// TIA Portal V20 export
FUNCTION_BLOCK "EventsPFE_Recipe"   // FB125, LAD
// stored: MemoryReserve 100, Namespace Unit1.Em7, SetENOAutomatically false
   VAR
      data : Array[1..100] of LReal;
   END_VAR
BEGIN

REGION Network 1: PDR Data21 Recipe - Hot Press Right Press Pressure
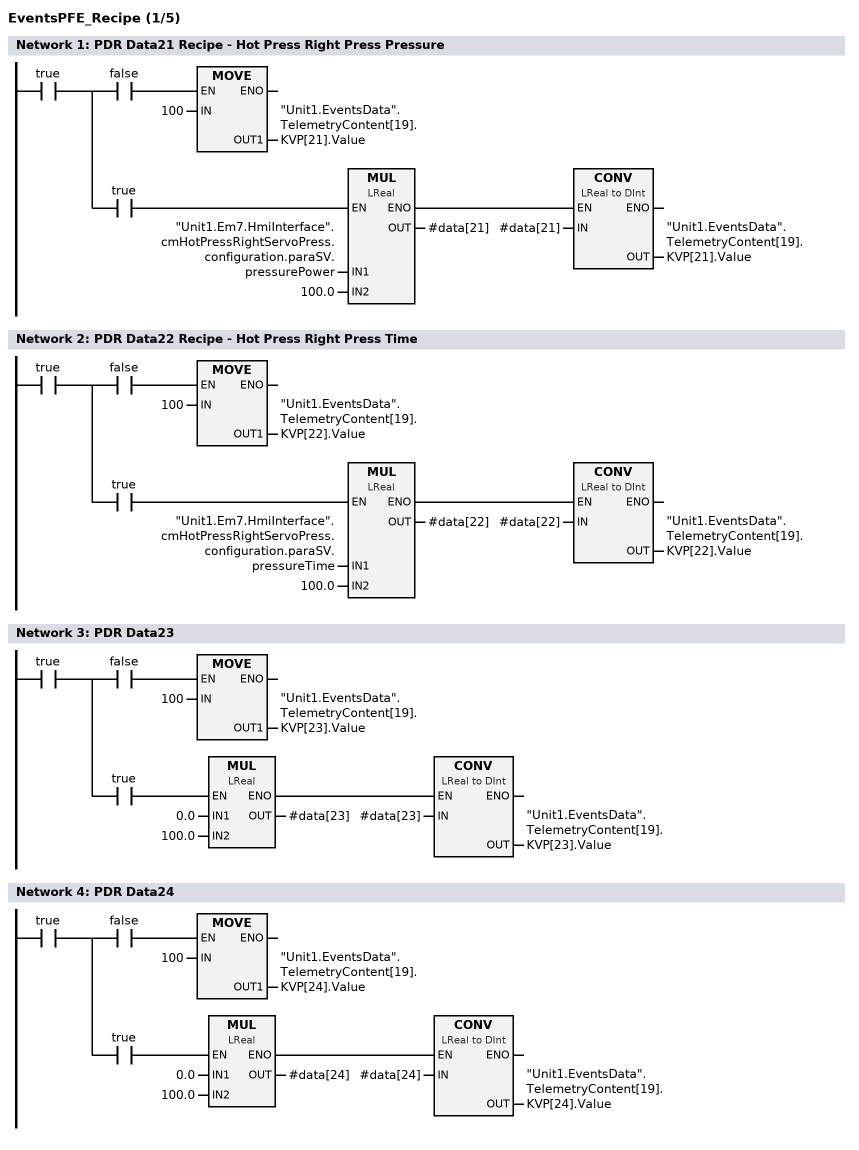
   RUNG wire#powerrail
      Contact( true )
      wire#w1
      Contact( false )
      Move(in := 100, out1 => "Unit1.EventsData".TelemetryContent[19].KVP[21].Value)
   END_RUNG
   RUNG wire#w1
      Contact( true )
      { S7_Templates := "SrcType := LReal" } Mul(in1 := "Unit1.Em7.HmiInterface".cmHotPressRightServoPress.configuration.paraSV.pressurePower, in2 := 100.0, out => #data[21])
      { S7_Templates := "[SrcType := LReal, DestType := DInt]" } Convert(in := #data[21], out => "Unit1.EventsData".TelemetryContent[19].KVP[21].Value)
   END_RUNG
   // the same network as SCL:
   IF true AND false THEN "Unit1.EventsData".TelemetryContent[19].KVP[21].Value := 100; END_IF;
   IF true AND true THEN
       #data[21] := "Unit1.Em7.HmiInterface".cmHotPressRightServoPress.configuration.paraSV.pressurePower * 100.0;
       "Unit1.EventsData".TelemetryContent[19].KVP[21].Value := LREAL_TO_DINT(#data[21]);
   END_IF;
END_REGION

REGION Network 2: PDR Data22 Recipe - Hot Press Right Press Time
   RUNG wire#powerrail
      Contact( true )
      wire#w1
      Contact( false )
      Move(in := 100, out1 => "Unit1.EventsData".TelemetryContent[19].KVP[22].Value)
   END_RUNG
   RUNG wire#w1
      Contact( true )
      { S7_Templates := "SrcType := LReal" } Mul(in1 := "Unit1.Em7.HmiInterface".cmHotPressRightServoPress.configuration.paraSV.pressureTime, in2 := 100.0, out => #data[22])
      { S7_Templates := "[SrcType := LReal, DestType := DInt]" } Convert(in := #data[22], out => "Unit1.EventsData".TelemetryContent[19].KVP[22].Value)
   END_RUNG
   // the same network as SCL:
   IF true AND false THEN "Unit1.EventsData".TelemetryContent[19].KVP[22].Value := 100; END_IF;
   IF true AND true THEN
       #data[22] := "Unit1.Em7.HmiInterface".cmHotPressRightServoPress.configuration.paraSV.pressureTime * 100.0;
       "Unit1.EventsData".TelemetryContent[19].KVP[22].Value := LREAL_TO_DINT(#data[22]);
   END_IF;
END_REGION

REGION Network 3: PDR Data23
   RUNG wire#powerrail
      Contact( true )
      wire#w1
      Contact( false )
      Move(in := 100, out1 => "Unit1.EventsData".TelemetryContent[19].KVP[23].Value)
   END_RUNG
   RUNG wire#w1
      Contact( true )
      { S7_Templates := "SrcType := LReal" } Mul(in1 := 0.0, in2 := 100.0, out => #data[23])
      { S7_Templates := "[SrcType := LReal, DestType := DInt]" } Convert(in := #data[23], out => "Unit1.EventsData".TelemetryContent[19].KVP[23].Value)
   END_RUNG
   // the same network as SCL:
   IF true AND false THEN "Unit1.EventsData".TelemetryContent[19].KVP[23].Value := 100; END_IF;
   IF true AND true THEN
       #data[23] := 0.0 * 100.0;
       "Unit1.EventsData".TelemetryContent[19].KVP[23].Value := LREAL_TO_DINT(#data[23]);
   END_IF;
END_REGION

REGION Network 4: PDR Data24
   RUNG wire#powerrail
      Contact( true )
      wire#w1
      Contact( false )
      Move(in := 100, out1 => "Unit1.EventsData".TelemetryContent[19].KVP[24].Value)
   END_RUNG
   RUNG wire#w1
      Contact( true )
      { S7_Templates := "SrcType := LReal" } Mul(in1 := 0.0, in2 := 100.0, out => #data[24])
      { S7_Templates := "[SrcType := LReal, DestType := DInt]" } Convert(in := #data[24], out => "Unit1.EventsData".TelemetryContent[19].KVP[24].Value)
   END_RUNG
   // the same network as SCL:
   IF true AND false THEN "Unit1.EventsData".TelemetryContent[19].KVP[24].Value := 100; END_IF;
   IF true AND true THEN
       #data[24] := 0.0 * 100.0;
       "Unit1.EventsData".TelemetryContent[19].KVP[24].Value := LREAL_TO_DINT(#data[24]);
   END_IF;
END_REGION

REGION Network 5: PDR Data25 Recipe - Hot Press Right Upper1 Temperature
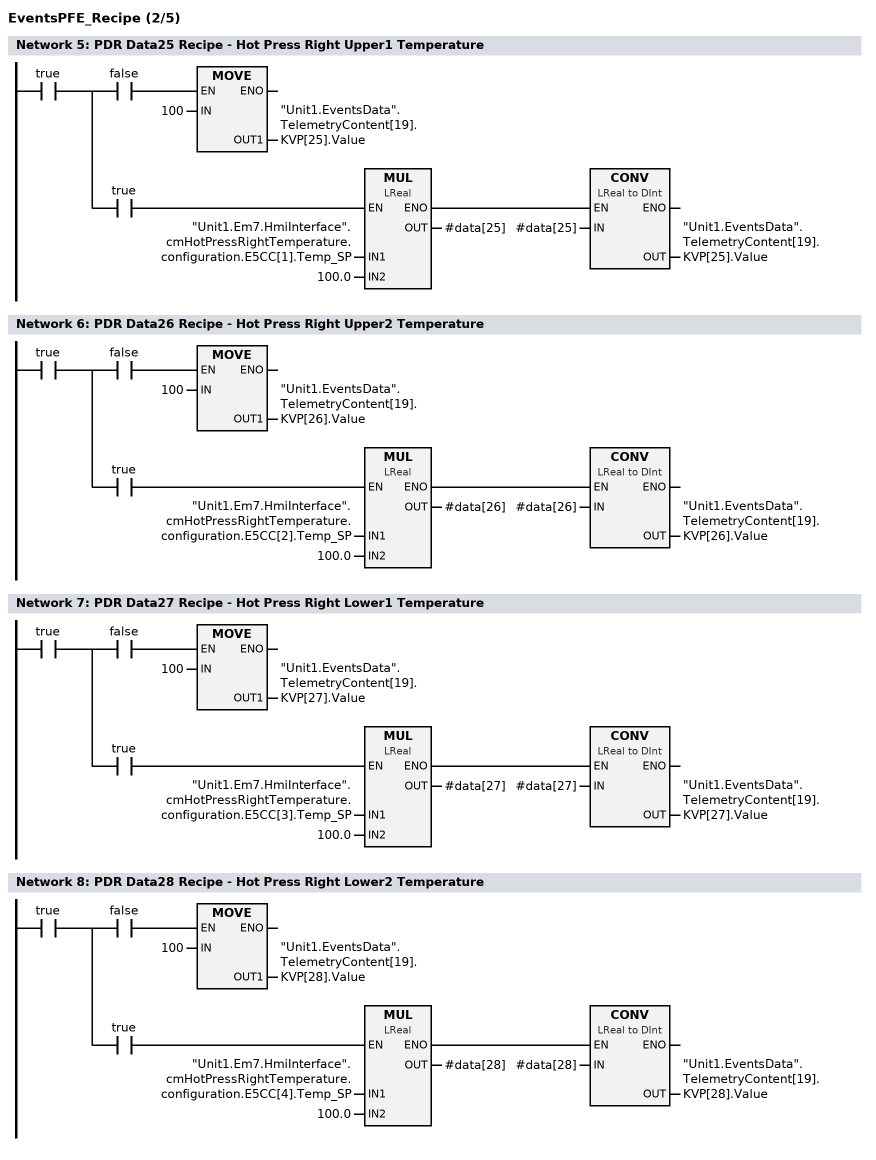
   RUNG wire#powerrail
      Contact( true )
      wire#w1
      Contact( false )
      Move(in := 100, out1 => "Unit1.EventsData".TelemetryContent[19].KVP[25].Value)
   END_RUNG
   RUNG wire#w1
      Contact( true )
      { S7_Templates := "SrcType := LReal" } Mul(in1 := "Unit1.Em7.HmiInterface".cmHotPressRightTemperature.configuration.E5CC[1].Temp_SP, in2 := 100.0, out => #data[25])
      { S7_Templates := "[SrcType := LReal, DestType := DInt]" } Convert(in := #data[25], out => "Unit1.EventsData".TelemetryContent[19].KVP[25].Value)
   END_RUNG
   // the same network as SCL:
   IF true AND false THEN "Unit1.EventsData".TelemetryContent[19].KVP[25].Value := 100; END_IF;
   IF true AND true THEN
       #data[25] := "Unit1.Em7.HmiInterface".cmHotPressRightTemperature.configuration.E5CC[1].Temp_SP * 100.0;
       "Unit1.EventsData".TelemetryContent[19].KVP[25].Value := LREAL_TO_DINT(#data[25]);
   END_IF;
END_REGION

REGION Network 6: PDR Data26 Recipe - Hot Press Right Upper2 Temperature
   RUNG wire#powerrail
      Contact( true )
      wire#w1
      Contact( false )
      Move(in := 100, out1 => "Unit1.EventsData".TelemetryContent[19].KVP[26].Value)
   END_RUNG
   RUNG wire#w1
      Contact( true )
      { S7_Templates := "SrcType := LReal" } Mul(in1 := "Unit1.Em7.HmiInterface".cmHotPressRightTemperature.configuration.E5CC[2].Temp_SP, in2 := 100.0, out => #data[26])
      { S7_Templates := "[SrcType := LReal, DestType := DInt]" } Convert(in := #data[26], out => "Unit1.EventsData".TelemetryContent[19].KVP[26].Value)
   END_RUNG
   // the same network as SCL:
   IF true AND false THEN "Unit1.EventsData".TelemetryContent[19].KVP[26].Value := 100; END_IF;
   IF true AND true THEN
       #data[26] := "Unit1.Em7.HmiInterface".cmHotPressRightTemperature.configuration.E5CC[2].Temp_SP * 100.0;
       "Unit1.EventsData".TelemetryContent[19].KVP[26].Value := LREAL_TO_DINT(#data[26]);
   END_IF;
END_REGION

REGION Network 7: PDR Data27 Recipe - Hot Press Right Lower1 Temperature
   RUNG wire#powerrail
      Contact( true )
      wire#w1
      Contact( false )
      Move(in := 100, out1 => "Unit1.EventsData".TelemetryContent[19].KVP[27].Value)
   END_RUNG
   RUNG wire#w1
      Contact( true )
      { S7_Templates := "SrcType := LReal" } Mul(in1 := "Unit1.Em7.HmiInterface".cmHotPressRightTemperature.configuration.E5CC[3].Temp_SP, in2 := 100.0, out => #data[27])
      { S7_Templates := "[SrcType := LReal, DestType := DInt]" } Convert(in := #data[27], out => "Unit1.EventsData".TelemetryContent[19].KVP[27].Value)
   END_RUNG
   // the same network as SCL:
   IF true AND false THEN "Unit1.EventsData".TelemetryContent[19].KVP[27].Value := 100; END_IF;
   IF true AND true THEN
       #data[27] := "Unit1.Em7.HmiInterface".cmHotPressRightTemperature.configuration.E5CC[3].Temp_SP * 100.0;
       "Unit1.EventsData".TelemetryContent[19].KVP[27].Value := LREAL_TO_DINT(#data[27]);
   END_IF;
END_REGION

REGION Network 8: PDR Data28 Recipe - Hot Press Right Lower2 Temperature
   RUNG wire#powerrail
      Contact( true )
      wire#w1
      Contact( false )
      Move(in := 100, out1 => "Unit1.EventsData".TelemetryContent[19].KVP[28].Value)
   END_RUNG
   RUNG wire#w1
      Contact( true )
      { S7_Templates := "SrcType := LReal" } Mul(in1 := "Unit1.Em7.HmiInterface".cmHotPressRightTemperature.configuration.E5CC[4].Temp_SP, in2 := 100.0, out => #data[28])
      { S7_Templates := "[SrcType := LReal, DestType := DInt]" } Convert(in := #data[28], out => "Unit1.EventsData".TelemetryContent[19].KVP[28].Value)
   END_RUNG
   // the same network as SCL:
   IF true AND false THEN "Unit1.EventsData".TelemetryContent[19].KVP[28].Value := 100; END_IF;
   IF true AND true THEN
       #data[28] := "Unit1.Em7.HmiInterface".cmHotPressRightTemperature.configuration.E5CC[4].Temp_SP * 100.0;
       "Unit1.EventsData".TelemetryContent[19].KVP[28].Value := LREAL_TO_DINT(#data[28]);
   END_IF;
END_REGION

REGION Network 9: PDR Data29 Recipe - Hot Press Right Lower3 Temperature
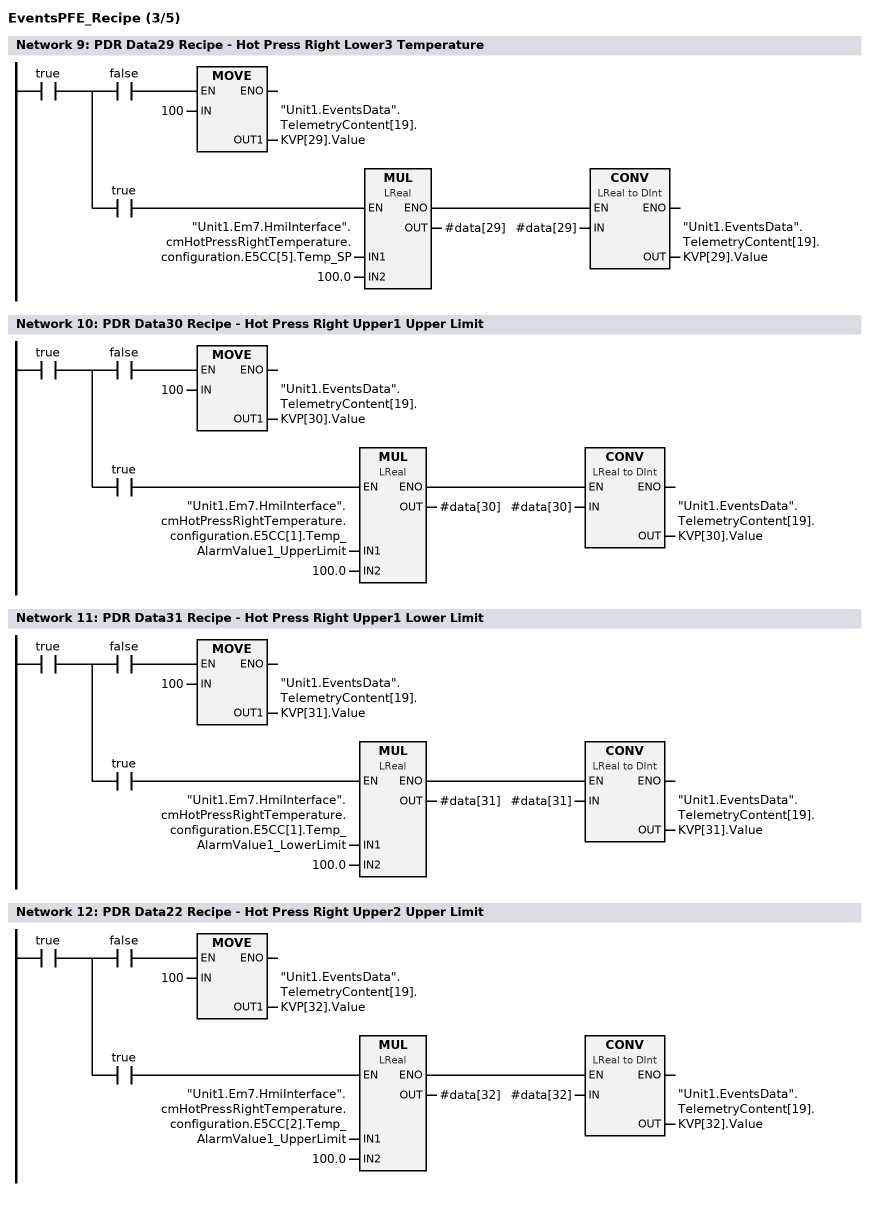
   RUNG wire#powerrail
      Contact( true )
      wire#w1
      Contact( false )
      Move(in := 100, out1 => "Unit1.EventsData".TelemetryContent[19].KVP[29].Value)
   END_RUNG
   RUNG wire#w1
      Contact( true )
      { S7_Templates := "SrcType := LReal" } Mul(in1 := "Unit1.Em7.HmiInterface".cmHotPressRightTemperature.configuration.E5CC[5].Temp_SP, in2 := 100.0, out => #data[29])
      { S7_Templates := "[SrcType := LReal, DestType := DInt]" } Convert(in := #data[29], out => "Unit1.EventsData".TelemetryContent[19].KVP[29].Value)
   END_RUNG
   // the same network as SCL:
   IF true AND false THEN "Unit1.EventsData".TelemetryContent[19].KVP[29].Value := 100; END_IF;
   IF true AND true THEN
       #data[29] := "Unit1.Em7.HmiInterface".cmHotPressRightTemperature.configuration.E5CC[5].Temp_SP * 100.0;
       "Unit1.EventsData".TelemetryContent[19].KVP[29].Value := LREAL_TO_DINT(#data[29]);
   END_IF;
END_REGION

REGION Network 10: PDR Data30 Recipe - Hot Press Right Upper1 Upper Limit
   RUNG wire#powerrail
      Contact( true )
      wire#w1
      Contact( false )
      Move(in := 100, out1 => "Unit1.EventsData".TelemetryContent[19].KVP[30].Value)
   END_RUNG
   RUNG wire#w1
      Contact( true )
      { S7_Templates := "SrcType := LReal" } Mul(in1 := "Unit1.Em7.HmiInterface".cmHotPressRightTemperature.configuration.E5CC[1].Temp_AlarmValue1_UpperLimit, in2 := 100.0, out => #data[30])
      { S7_Templates := "[SrcType := LReal, DestType := DInt]" } Convert(in := #data[30], out => "Unit1.EventsData".TelemetryContent[19].KVP[30].Value)
   END_RUNG
   // the same network as SCL:
   IF true AND false THEN "Unit1.EventsData".TelemetryContent[19].KVP[30].Value := 100; END_IF;
   IF true AND true THEN
       #data[30] := "Unit1.Em7.HmiInterface".cmHotPressRightTemperature.configuration.E5CC[1].Temp_AlarmValue1_UpperLimit * 100.0;
       "Unit1.EventsData".TelemetryContent[19].KVP[30].Value := LREAL_TO_DINT(#data[30]);
   END_IF;
END_REGION

REGION Network 11: PDR Data31 Recipe - Hot Press Right Upper1 Lower Limit
   RUNG wire#powerrail
      Contact( true )
      wire#w1
      Contact( false )
      Move(in := 100, out1 => "Unit1.EventsData".TelemetryContent[19].KVP[31].Value)
   END_RUNG
   RUNG wire#w1
      Contact( true )
      { S7_Templates := "SrcType := LReal" } Mul(in1 := "Unit1.Em7.HmiInterface".cmHotPressRightTemperature.configuration.E5CC[1].Temp_AlarmValue1_LowerLimit, in2 := 100.0, out => #data[31])
      { S7_Templates := "[SrcType := LReal, DestType := DInt]" } Convert(in := #data[31], out => "Unit1.EventsData".TelemetryContent[19].KVP[31].Value)
   END_RUNG
   // the same network as SCL:
   IF true AND false THEN "Unit1.EventsData".TelemetryContent[19].KVP[31].Value := 100; END_IF;
   IF true AND true THEN
       #data[31] := "Unit1.Em7.HmiInterface".cmHotPressRightTemperature.configuration.E5CC[1].Temp_AlarmValue1_LowerLimit * 100.0;
       "Unit1.EventsData".TelemetryContent[19].KVP[31].Value := LREAL_TO_DINT(#data[31]);
   END_IF;
END_REGION

REGION Network 12: PDR Data22 Recipe - Hot Press Right Upper2 Upper Limit
   RUNG wire#powerrail
      Contact( true )
      wire#w1
      Contact( false )
      Move(in := 100, out1 => "Unit1.EventsData".TelemetryContent[19].KVP[32].Value)
   END_RUNG
   RUNG wire#w1
      Contact( true )
      { S7_Templates := "SrcType := LReal" } Mul(in1 := "Unit1.Em7.HmiInterface".cmHotPressRightTemperature.configuration.E5CC[2].Temp_AlarmValue1_UpperLimit, in2 := 100.0, out => #data[32])
      { S7_Templates := "[SrcType := LReal, DestType := DInt]" } Convert(in := #data[32], out => "Unit1.EventsData".TelemetryContent[19].KVP[32].Value)
   END_RUNG
   // the same network as SCL:
   IF true AND false THEN "Unit1.EventsData".TelemetryContent[19].KVP[32].Value := 100; END_IF;
   IF true AND true THEN
       #data[32] := "Unit1.Em7.HmiInterface".cmHotPressRightTemperature.configuration.E5CC[2].Temp_AlarmValue1_UpperLimit * 100.0;
       "Unit1.EventsData".TelemetryContent[19].KVP[32].Value := LREAL_TO_DINT(#data[32]);
   END_IF;
END_REGION

REGION Network 13: PDR Data33 Recipe - Hot Press Right Upper2 Lower Limit
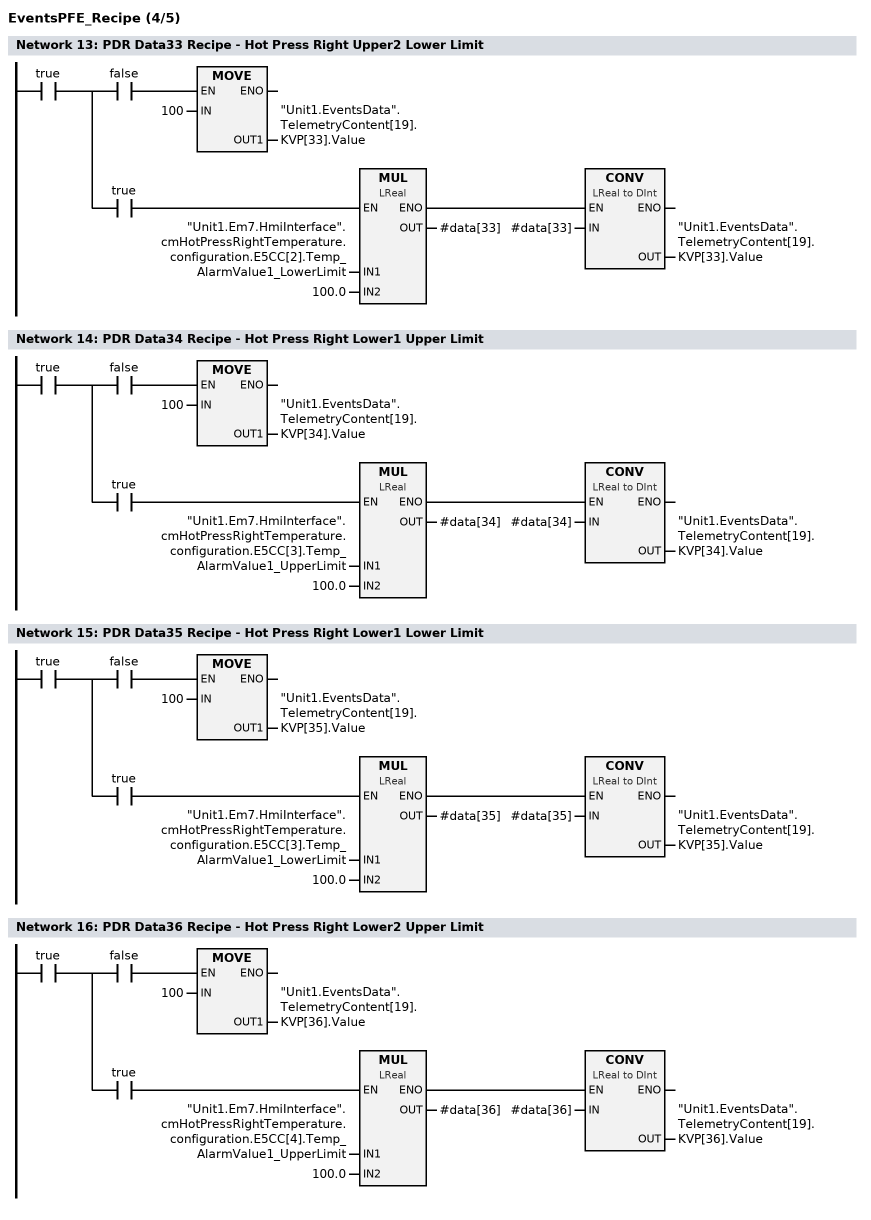
   RUNG wire#powerrail
      Contact( true )
      wire#w1
      Contact( false )
      Move(in := 100, out1 => "Unit1.EventsData".TelemetryContent[19].KVP[33].Value)
   END_RUNG
   RUNG wire#w1
      Contact( true )
      { S7_Templates := "SrcType := LReal" } Mul(in1 := "Unit1.Em7.HmiInterface".cmHotPressRightTemperature.configuration.E5CC[2].Temp_AlarmValue1_LowerLimit, in2 := 100.0, out => #data[33])
      { S7_Templates := "[SrcType := LReal, DestType := DInt]" } Convert(in := #data[33], out => "Unit1.EventsData".TelemetryContent[19].KVP[33].Value)
   END_RUNG
   // the same network as SCL:
   IF true AND false THEN "Unit1.EventsData".TelemetryContent[19].KVP[33].Value := 100; END_IF;
   IF true AND true THEN
       #data[33] := "Unit1.Em7.HmiInterface".cmHotPressRightTemperature.configuration.E5CC[2].Temp_AlarmValue1_LowerLimit * 100.0;
       "Unit1.EventsData".TelemetryContent[19].KVP[33].Value := LREAL_TO_DINT(#data[33]);
   END_IF;
END_REGION

REGION Network 14: PDR Data34 Recipe - Hot Press Right Lower1 Upper Limit
   RUNG wire#powerrail
      Contact( true )
      wire#w1
      Contact( false )
      Move(in := 100, out1 => "Unit1.EventsData".TelemetryContent[19].KVP[34].Value)
   END_RUNG
   RUNG wire#w1
      Contact( true )
      { S7_Templates := "SrcType := LReal" } Mul(in1 := "Unit1.Em7.HmiInterface".cmHotPressRightTemperature.configuration.E5CC[3].Temp_AlarmValue1_UpperLimit, in2 := 100.0, out => #data[34])
      { S7_Templates := "[SrcType := LReal, DestType := DInt]" } Convert(in := #data[34], out => "Unit1.EventsData".TelemetryContent[19].KVP[34].Value)
   END_RUNG
   // the same network as SCL:
   IF true AND false THEN "Unit1.EventsData".TelemetryContent[19].KVP[34].Value := 100; END_IF;
   IF true AND true THEN
       #data[34] := "Unit1.Em7.HmiInterface".cmHotPressRightTemperature.configuration.E5CC[3].Temp_AlarmValue1_UpperLimit * 100.0;
       "Unit1.EventsData".TelemetryContent[19].KVP[34].Value := LREAL_TO_DINT(#data[34]);
   END_IF;
END_REGION

REGION Network 15: PDR Data35 Recipe - Hot Press Right Lower1 Lower Limit
   RUNG wire#powerrail
      Contact( true )
      wire#w1
      Contact( false )
      Move(in := 100, out1 => "Unit1.EventsData".TelemetryContent[19].KVP[35].Value)
   END_RUNG
   RUNG wire#w1
      Contact( true )
      { S7_Templates := "SrcType := LReal" } Mul(in1 := "Unit1.Em7.HmiInterface".cmHotPressRightTemperature.configuration.E5CC[3].Temp_AlarmValue1_LowerLimit, in2 := 100.0, out => #data[35])
      { S7_Templates := "[SrcType := LReal, DestType := DInt]" } Convert(in := #data[35], out => "Unit1.EventsData".TelemetryContent[19].KVP[35].Value)
   END_RUNG
   // the same network as SCL:
   IF true AND false THEN "Unit1.EventsData".TelemetryContent[19].KVP[35].Value := 100; END_IF;
   IF true AND true THEN
       #data[35] := "Unit1.Em7.HmiInterface".cmHotPressRightTemperature.configuration.E5CC[3].Temp_AlarmValue1_LowerLimit * 100.0;
       "Unit1.EventsData".TelemetryContent[19].KVP[35].Value := LREAL_TO_DINT(#data[35]);
   END_IF;
END_REGION

REGION Network 16: PDR Data36 Recipe - Hot Press Right Lower2 Upper Limit
   RUNG wire#powerrail
      Contact( true )
      wire#w1
      Contact( false )
      Move(in := 100, out1 => "Unit1.EventsData".TelemetryContent[19].KVP[36].Value)
   END_RUNG
   RUNG wire#w1
      Contact( true )
      { S7_Templates := "SrcType := LReal" } Mul(in1 := "Unit1.Em7.HmiInterface".cmHotPressRightTemperature.configuration.E5CC[4].Temp_AlarmValue1_UpperLimit, in2 := 100.0, out => #data[36])
      { S7_Templates := "[SrcType := LReal, DestType := DInt]" } Convert(in := #data[36], out => "Unit1.EventsData".TelemetryContent[19].KVP[36].Value)
   END_RUNG
   // the same network as SCL:
   IF true AND false THEN "Unit1.EventsData".TelemetryContent[19].KVP[36].Value := 100; END_IF;
   IF true AND true THEN
       #data[36] := "Unit1.Em7.HmiInterface".cmHotPressRightTemperature.configuration.E5CC[4].Temp_AlarmValue1_UpperLimit * 100.0;
       "Unit1.EventsData".TelemetryContent[19].KVP[36].Value := LREAL_TO_DINT(#data[36]);
   END_IF;
END_REGION

REGION Network 17: PDR Data37 Recipe - Hot Press Right Lower2 Lower Limit
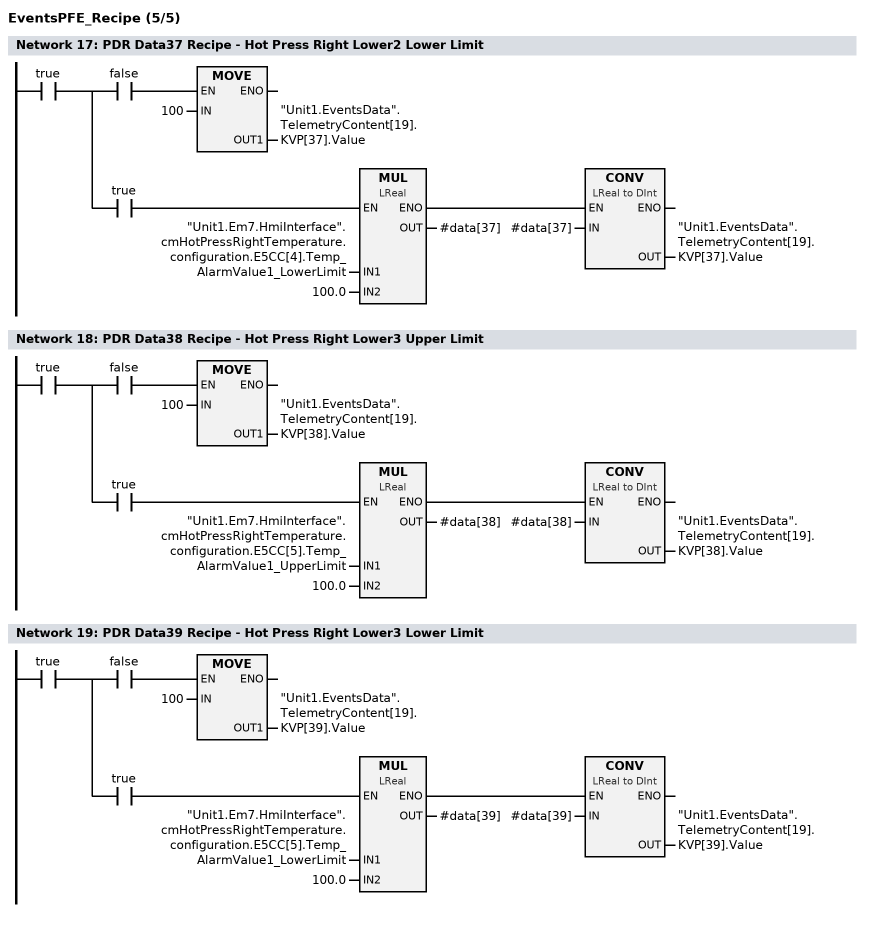
   RUNG wire#powerrail
      Contact( true )
      wire#w1
      Contact( false )
      Move(in := 100, out1 => "Unit1.EventsData".TelemetryContent[19].KVP[37].Value)
   END_RUNG
   RUNG wire#w1
      Contact( true )
      { S7_Templates := "SrcType := LReal" } Mul(in1 := "Unit1.Em7.HmiInterface".cmHotPressRightTemperature.configuration.E5CC[4].Temp_AlarmValue1_LowerLimit, in2 := 100.0, out => #data[37])
      { S7_Templates := "[SrcType := LReal, DestType := DInt]" } Convert(in := #data[37], out => "Unit1.EventsData".TelemetryContent[19].KVP[37].Value)
   END_RUNG
   // the same network as SCL:
   IF true AND false THEN "Unit1.EventsData".TelemetryContent[19].KVP[37].Value := 100; END_IF;
   IF true AND true THEN
       #data[37] := "Unit1.Em7.HmiInterface".cmHotPressRightTemperature.configuration.E5CC[4].Temp_AlarmValue1_LowerLimit * 100.0;
       "Unit1.EventsData".TelemetryContent[19].KVP[37].Value := LREAL_TO_DINT(#data[37]);
   END_IF;
END_REGION

REGION Network 18: PDR Data38 Recipe - Hot Press Right Lower3 Upper Limit
   RUNG wire#powerrail
      Contact( true )
      wire#w1
      Contact( false )
      Move(in := 100, out1 => "Unit1.EventsData".TelemetryContent[19].KVP[38].Value)
   END_RUNG
   RUNG wire#w1
      Contact( true )
      { S7_Templates := "SrcType := LReal" } Mul(in1 := "Unit1.Em7.HmiInterface".cmHotPressRightTemperature.configuration.E5CC[5].Temp_AlarmValue1_UpperLimit, in2 := 100.0, out => #data[38])
      { S7_Templates := "[SrcType := LReal, DestType := DInt]" } Convert(in := #data[38], out => "Unit1.EventsData".TelemetryContent[19].KVP[38].Value)
   END_RUNG
   // the same network as SCL:
   IF true AND false THEN "Unit1.EventsData".TelemetryContent[19].KVP[38].Value := 100; END_IF;
   IF true AND true THEN
       #data[38] := "Unit1.Em7.HmiInterface".cmHotPressRightTemperature.configuration.E5CC[5].Temp_AlarmValue1_UpperLimit * 100.0;
       "Unit1.EventsData".TelemetryContent[19].KVP[38].Value := LREAL_TO_DINT(#data[38]);
   END_IF;
END_REGION

REGION Network 19: PDR Data39 Recipe - Hot Press Right Lower3 Lower Limit
   RUNG wire#powerrail
      Contact( true )
      wire#w1
      Contact( false )
      Move(in := 100, out1 => "Unit1.EventsData".TelemetryContent[19].KVP[39].Value)
   END_RUNG
   RUNG wire#w1
      Contact( true )
      { S7_Templates := "SrcType := LReal" } Mul(in1 := "Unit1.Em7.HmiInterface".cmHotPressRightTemperature.configuration.E5CC[5].Temp_AlarmValue1_LowerLimit, in2 := 100.0, out => #data[39])
      { S7_Templates := "[SrcType := LReal, DestType := DInt]" } Convert(in := #data[39], out => "Unit1.EventsData".TelemetryContent[19].KVP[39].Value)
   END_RUNG
   // the same network as SCL:
   IF true AND false THEN "Unit1.EventsData".TelemetryContent[19].KVP[39].Value := 100; END_IF;
   IF true AND true THEN
       #data[39] := "Unit1.Em7.HmiInterface".cmHotPressRightTemperature.configuration.E5CC[5].Temp_AlarmValue1_LowerLimit * 100.0;
       "Unit1.EventsData".TelemetryContent[19].KVP[39].Value := LREAL_TO_DINT(#data[39]);
   END_IF;
END_REGION
END_FUNCTION_BLOCK
